(* PLC project TON timer FBD, react-plc-diagram PLCopen XML test fixtures 0.1.0 *)
(* stored: creationDateTime 2026-08-12T00:00:00Z, modificationDateTime 2026-08-12T00:00:00Z *)

PROGRAM DelayedFan
  VAR
    Enable : BOOL;
    Delay : TIME := T#3s;
    Fan : BOOL;
    FanTimer : TON;
  END_VAR

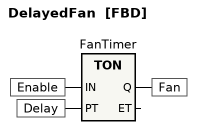
(* FBD diagram, written out as Structured Text *)
FanTimer(IN := Enable, PT := Delay);
Fan := FanTimer.Q;
END_PROGRAM
